# EPICS substitutions: iocBoot/iocTomoStream/tomoStream.substitutions
file "$(TOP)/db/tomoStream.template"
{
pattern
{  P,      R, TOMO_SCAN, IMAGE_P, DARK_PVA, FLAT_PVA, RECON_PVA}
{2bmb:, TomoStream:, 2bmb:TomoScan:, 2bmb:TomoScan:PvaPluginPVPrefix, 2bmb:TomoScan:StreamDarkFields, 2bmb:TomoScan:StreamFlatFields, 2bmb:TomoStream:StreamRecon}
}
